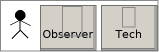
VISUALIZATION VISU_OperatorStatus  // 159x52
VAR_IN_OUT
	status : OperatorStatus;
	process : ChangeOperatorStateProcess;
END_VAR
    Line (20,30) (20,20)
    Line (12,38) (20,30)
    Line (28,38) (20,30)
    Line (20,20) (10,25)
    Line (20,20) (30,25)
    Ellipse (15,10 10x10)
    Button (101,5 56x45), "Tech", input disabled if: process.statuses.enabledStatus.disabled
        OnMouseClick: execute { process.set.state := OperatorStates.TECH; process.do_request := TRUE; }
        OnMouseDown: execute {  }
    Frame (122,7 13x20)
        shows VISU_State_gray_orange(state := status.tech)
        OnMouseClick: execute { process.set.state := OperatorStates.TECH; process.do_request := TRUE; }
    Button (40,5 56x45), "Observer", input disabled if: process.statuses.enabledStatus.disabled
        OnMouseClick: execute { process.set.state := OperatorStates.OBSERVER; process.do_request := TRUE; }
        OnMouseDown: execute {  }
    Frame (62,6 20x30)
        shows VISU_State_gray_green(state := status.observer)
        OnMouseClick: execute { process.set.state := OperatorStates.OBSERVER; process.do_request := TRUE; }
END_VISUALIZATION

(* stored: Version 1.1.0.1, ProductVersion 3.1.4019.2
   Visu VISU_OperatorStatus: Id {c604b407-7f50-40f2-85d5-235682e33698} *)
